// Mitsubishi GX Works2 project: game   PLC: FX3U/FX3UC

// task Task_01 (event TRUE, interval 0, priority 31): POU_01

PROGRAM POU_01
VAR
  wstep : INT;
  rand : INT;
  won : ARRAY [0..7] OF INT;
  team1 : INT;
  team2 : INT;
  DRAW_team1 : DRAW;
  DRAW_team2 : DRAW;
  TON_RAND : TON;
  TON_1 : TON;
  TON_2 : TON;
  ii : INT;
  winner : BOOL;
  R_TRIG_1 : R_TRIG;
  R_TRIG_2 : R_TRIG;
  TON_team1 : TON;
  TON_team2 : TON;
  TON_show : TON;
  TON_win : TON;
  TON_switch1 : TON;
  TON_switch2 : TON;
END_VAR
M99 := 
(*Y*)
Y0 AND Y12 AND Y13 AND

Y1 AND Y2 AND Y3 AND 
Y4 AND Y5 AND Y6 AND
Y7 AND Y10 AND Y11 AND 
 
(*X*)		 
X0 AND X12 AND
X1 AND X2  AND X3 AND 
X4 AND X5 AND X6 AND 
X7 AND X10 AND X11;

IF M8002 OR X12 THEN
	wstep := 0;
END_IF;

IF wstep <> 0 THEN 
	(*win*)
	IF 		
		(Y1 AND Y5 AND Y11) OR (Y3 AND Y5 AND Y7) OR 
		(Y1 AND Y2 AND Y3) OR (Y4 AND Y5 AND Y6) OR (Y7 AND Y10 AND Y11) OR
		(Y1 AND Y4 AND Y7) OR (Y2 AND Y5 AND Y10) OR (Y3 AND Y6 AND Y11)
	THEN
		winner := Y12;
		wstep := 70; 
		ZRST(TRUE, Y0, Y17);
	END_IF;
	
	(*pease*)
	IF  Y1 AND Y2 AND Y3 AND Y4 AND Y5 AND Y6 AND Y7 AND Y10 AND Y11 THEN
		wstep := 70;
		ZRST(TRUE, Y0, Y17);
	END_IF;
END_IF;

CASE  wstep  OF
	
	(*default*)
	0:
	ZRST(TRUE, Y0, Y17);
	K4Y0 := 4095;
	team1 := 1024;
	team2 := 2048;
	TON_1( IN := NOT TON_1.Q, PT := T#2s);
	IF TON_1.Q THEN
		K4Y0 := 0;
		wstep := 20;
	END_IF;
	
	(*set who start first and ready to start*)
	20:
	TON_RAND( IN := NOT TON_RAND.Q, PT := T#50ms); (*rand*)
	INC(TRUE, rand);
	IF rand = 10 THEN
		rand := 0;
	END_IF;
	IF X0 THEN
		IF (rand MOD 2) = 1 THEN
			wstep := 40;
		ELSE
			wstep := 50;
		END_IF;
	END_IF;
	
	(*team1*)
	40:
	TON_switch1(IN := NOT TON_switch2.Q, PT := T#2s);
	TON_switch2(IN := TON_switch1.Q, PT := T#1s);
	IF TON_switch1.Q AND ((NOT (K4X0 >= 2)) OR DRAW_team1.resultB) THEN
		K4Y0 := team2;
	ELSE 
		K4Y0 := team1;
	END_IF;
	DRAW_team1(IN := TRUE, teamA := team1, teamB := team2);
	IF DRAW_team1.resultA THEN
		K4Y0 := team1 + K4X0;
		TON_team1(IN := NOT TON_team1.Q, PT := T#2s);
		IF TON_team1.Q THEN
			team1 := team1 + K4X0;
			DRAW_team1(IN := FALSE);
			wstep := 50;
		END_IF;
	ELSIF DRAW_team1.resultB THEN 
		Y0 := M8013;
	END_IF;
	
	(*team2*)
	50:
	TON_switch1(IN := NOT TON_switch2.Q, PT := T#2s);
	TON_switch2(IN := TON_switch1.Q, PT := T#1s);
	IF TON_switch1.Q AND ((NOT (K4X0 >= 2)) OR DRAW_team2.resultB) THEN
		K4Y0 := team1;
	ELSE 
		K4Y0 := team2;
	END_IF;
	DRAW_team2(IN := TRUE, teamA := team1, teamB := team2);
	IF DRAW_team2.resultA THEN
		K4Y0 := team2 + K4X0;
		TON_team2(IN :=  NOT TON_team2.Q, PT := T#2s);
		IF TON_team2.Q THEN
			team2 := team2 + K4X0;
			DRAW_team2(IN := FALSE);
			wstep := 40;	
		END_IF;
	ELSIF DRAW_team2.resultB THEN
			Y0 := M8013;
	END_IF;
	
	(*win*)
	60:
	IF Y12 THEN
		Y12 := M8013;
	ELSE
		Y13 := M8013;
	END_IF;
	
	TON_win(IN := NOT TON_win.Q, PT := T#5s);
	IF TON_win.Q THEN
		wstep := 0;
	END_IF;
	
	(*pease*)
	70:
	INC(TRUE, K4Y0);
	wstep := 71;
	
	71:
	R_TRIG_1(_CLK:= M8012);
	IF R_TRIG_1.Q THEN
		ROL(TRUE, 1, K4Y0);
	END_IF;
	
	IF Y13 THEN
		wstep := 72;
	END_IF;
	
	72:
	R_TRIG_2(_CLK:= M8012);
	IF R_TRIG_2.Q THEN
		ROR(TRUE, 1, K4Y0);
	END_IF;
	
	IF Y0 THEN
		wstep := 0;
	END_IF;
END_CASE;
END_PROGRAM

FUNCTION_BLOCK DRAW
VAR_INPUT
  IN : BOOL;
END_VAR
VAR_OUTPUT
  resultA : BOOL;
  resultB : BOOL;
END_VAR
VAR_INPUT
  teamA : INT;
  teamB : INT;
END_VAR
VAR_OUTPUT
  result_team : INT;
END_VAR
VAR
  overlap : BOOL;
END_VAR
IF IN THEN
	D0 := K4X0; (*X*)
	D2 := teamA; (*Y*)
	D3 := teamB;
	D1 := 0;
	IF D0 > 1 AND D0 <= 512 THEN 
		WHILE D0 <> 0 DO (*get power*)
			D0 := D0 / 2;
			INC(TRUE, D1); 
		END_WHILE;
		DEC(TRUE, D1);
		ROR(TRUE, D1 , D2); (*if teamA had been trigged*)
		ROR(TRUE, D1 , D3); (*if teamB had been trigged*)
		overlap := (D2 MOD 2 = 0) AND (D3 MOD 2 = 0);
		resultA := overlap;
		resultB := NOT overlap;
	ELSE
		resultA := FALSE;
		resultB := FALSE;
	END_IF;
ELSE
	resultA := FALSE;
	resultB := FALSE;
END_IF;
END_FUNCTION_BLOCK
